(* IEC 61131-3 sources: AXOpen/src/components.cognex.vision/app/src/IO/PLC_LINE, 7 files *)

(* ---- HwIdentifiers.st ---- *)
TYPE
    HwIdentifiers : WORD
    (
        PROFINET_IO_System_HwID :=	WORD#256,
        is7600_HwID :=	WORD#259,
        is7600_Acquisition_Control_Acquisition_Control_HwID :=	WORD#269,
        is7600_Acquisition_Status_Acquisition_Status_HwID :=	WORD#265,
        is7600_Command_Control_Command_Control_HwID :=	WORD#266,
        is7600_Inspection_Control_Inspection_Control_HwID :=	WORD#268,
        is7600_Inspection_Status_Inspection_Status_HwID :=	WORD#264,
        is7600_Rack_HwID :=	WORD#260,
        is7600_Result_Data_64_bytes_Results___64_bytes_HwID :=	WORD#262,
        is7600_SoftEvent_Control_SoftEvent_Control_HwID :=	WORD#267,
        is7600_User_Data_64_bytes_User_Data___64_bytes_HwID :=	WORD#263,
        is7600_is7600_HwID :=	WORD#261,
        is7600_is7600_In_Sight_IS79XX_IS75XX_CC_B_HwID :=	WORD#270,
        is7600_is7600_profinet_HwID :=	WORD#257,
        is7600_is7600_profinet_Port_1_HwID :=	WORD#258,
        plc_line_HwID :=	WORD#32,
        plc_line_Rail_0_HwID :=	WORD#297,
        plc_line_plc_line_HwID :=	WORD#48,
        plc_line_plc_line__plc_line_HwID :=	WORD#49,
        plc_line_plc_line_CPU_display_1_HwID :=	WORD#54,
        plc_line_plc_line_CPU_exec_unit_1_HwID :=	WORD#52,
        plc_line_plc_line_Card_reader_writer_1_HwID :=	WORD#51,
        plc_line_plc_line_DP_interface_1_HwID :=	WORD#60,
        plc_line_plc_line_LicenseManager_1_HwID :=	WORD#42,
        plc_line_plc_line_OPC_UA_1_HwID :=	WORD#117,
        plc_line_plc_line_PROFINET_interface_2_HwID :=	WORD#72,
        plc_line_plc_line_PROFINET_interface_2_Port_1_HwID :=	WORD#73,
        plc_line_plc_line_Virtual_communication_interface_HwID :=	WORD#135,
        plc_line_plc_line_plc_line_HwID :=	WORD#50,
        plc_line_plc_line_profinet_x1_HwID :=	WORD#64,
        plc_line_plc_line_profinet_x1_Port1_HwID :=	WORD#65,
        plc_line_plc_line_profinet_x1_Port2_HwID :=	WORD#66,
        reader_st1_HwID :=	WORD#286,
        reader_st1_Acquisition_Control_Acquisition_Control_HwID :=	WORD#295,
        reader_st1_Acquisition_Status_Acquisition_Status_HwID :=	WORD#294,
        reader_st1_Rack_HwID :=	WORD#287,
        reader_st1_Result_Data_128_bytes_Result_Data___128_bytes_HwID :=	WORD#289,
        reader_st1_Results_Control_Results_Control_HwID :=	WORD#293,
        reader_st1_Results_Status_Results_Status_HwID :=	WORD#292,
        reader_st1_Soft_Event_Control_Soft_Event_Control_HwID :=	WORD#291,
        reader_st1_User_Data_128_bytes_User_Data___128_bytes_HwID :=	WORD#290,
        reader_st1_reader_st1_HwID :=	WORD#288,
        reader_st1_reader_st1_DataMan_280_CC_B_HwID :=	WORD#296,
        reader_st1_reader_st1_profinet_HwID :=	WORD#284,
        reader_st1_reader_st1_profinet_Port_1_HwID :=	WORD#285,
        reader_st2_HwID :=	WORD#273,
        reader_st2_Acquisition_Control_Acquisition_Control_HwID :=	WORD#282,
        reader_st2_Acquisition_Status_Acquisition_Status_HwID :=	WORD#281,
        reader_st2_Rack_HwID :=	WORD#274,
        reader_st2_Result_Data_64_bytes_Result_Data___64_bytes_HwID :=	WORD#276,
        reader_st2_Results_Control_Results_Control_HwID :=	WORD#280,
        reader_st2_Results_Status_Results_Status_HwID :=	WORD#279,
        reader_st2_Soft_Event_Control_Soft_Event_Control_HwID :=	WORD#278,
        reader_st2_User_Data_64_bytes_User_Data___64_bytes_HwID :=	WORD#277,
        reader_st2_reader_st2_HwID :=	WORD#275,
        reader_st2_reader_st2_DataMan_300_HwID :=	WORD#283,
        reader_st2_reader_st2_profinet_HwID :=	WORD#271,
        reader_st2_reader_st2_profinet_Port_1_HwID :=	WORD#272,

        NONE := WORD#0
    );
END_TYPE

(* ---- HwInputs.st ---- *)
TYPE
	HwInputs : STRUCT
		_10a1_Acquisition_Status_1 AT %B82 : ARRAY[0..2] OF BYTE;
		_10a1_Results_Status_1 AT %B85 : BYTE;
		_10a1_Soft_Event_Control_1 AT %B86 : BYTE;
		_10a1_Result_Data_128_bytes_1 AT %B87 : ARRAY[0..135] OF BYTE;
		reader_st2_Acquisition_Status_1 AT %B300 : ARRAY[0..2] OF BYTE;
		reader_st2_Results_Status_1 AT %B303 : BYTE;
		reader_st2_Soft_Event_Control_1 AT %B304 : BYTE;
		reader_st2_Result_Data_64_bytes_1 AT %B305 : ARRAY[0..71] OF BYTE;
		// _7600_Acquisition_Status_1 AT %B0 : ARRAY[0..2] OF BYTE;
		// _7600_Inspection_Status_1 AT %B3 : DWORD;
		// _7600_Command_Control_1 AT %B7 : WORD;
		// _7600_SoftEvent_Control_1 AT %B9 : BYTE;
		// _7600_Results_64_bytes_1 AT %B10 : ARRAY[0..67] OF BYTE;
	END_STRUCT;
END_TYPE

(* ---- HwOutputs.st ---- *)
TYPE
	HwOutputs : STRUCT
		_10a1_Acquisition_Control_1 AT %B72 : BYTE;
		_10a1_Results_Control_1 AT %B73 : BYTE;
		_10a1_Soft_Event_Control_1 AT %B74 : BYTE;
		_10a1_User_Data_128_bytes_1 AT %B75 : ARRAY[0..131] OF BYTE;
		reader_st2_Acquisition_Control_1 AT %B300 : BYTE;
		reader_st2_Results_Control_1 AT %B301 : BYTE;
		reader_st2_Soft_Event_Control_1 AT %B302 : BYTE;
		reader_st2_User_Data_64_bytes_1 AT %B303 : ARRAY[0..67] OF BYTE;
		// _7600_Acquisition_Control_1 AT %B0 : BYTE;
		// _7600_Inspection_Control_1 AT %B1 : BYTE;
		// _7600_Command_Control_1 AT %B2 : WORD;
		// _7600_SoftEvent_Control_1 AT %B4 : BYTE;
		// _7600_User_Data_64_bytes_1 AT %B5 : ARRAY[0..63] OF BYTE;
	END_STRUCT;
END_TYPE

(* ---- PlcInputs.st ---- *)
TYPE
	PlcInputs : STRUCT
		_10a1_Acquisition_Status_1 : ARRAY[0..2] OF BYTE;
		_10a1_Results_Status_1 : BYTE;
		_10a1_Soft_Event_Control_1 : BYTE;
		_10a1_Result_Data_128_bytes_1 : ARRAY[0..135] OF BYTE;
		reader_st2_Acquisition_Status_1 : ARRAY[0..2] OF BYTE;
		reader_st2_Results_Status_1 : BYTE;
		reader_st2_Soft_Event_Control_1 : BYTE;
		reader_st2_Result_Data_64_bytes_1 : ARRAY[0..71] OF BYTE;
		// _7600_Acquisition_Status_1 : ARRAY[0..2] OF BYTE;
		// _7600_Inspection_Status_1 : DWORD;
		// _7600_Command_Control_1 : WORD;
		// _7600_SoftEvent_Control_1 : BYTE;
		// _7600_Results_64_bytes_1 : ARRAY[0..67] OF BYTE;
	END_STRUCT;
END_TYPE

(* ---- PlcOutputs.st ---- *)
TYPE
	PlcOutputs : STRUCT
		_10a1_Acquisition_Control_1 : BYTE;
		_10a1_Results_Control_1 : BYTE;
		_10a1_Soft_Event_Control_1 : BYTE;
		_10a1_User_Data_128_bytes_1 : ARRAY[0..131] OF BYTE;
		reader_st2_Acquisition_Control_1 : BYTE;
		reader_st2_Results_Control_1 : BYTE;
		reader_st2_Soft_Event_Control_1 : BYTE;
		reader_st2_User_Data_64_bytes_1 : ARRAY[0..67] OF BYTE;
		// _7600_Acquisition_Control_1 : BYTE;
		// _7600_Inspection_Control_1 : BYTE;
		// _7600_Command_Control_1 : WORD;
		// _7600_SoftEvent_Control_1 : BYTE;
		// _7600_User_Data_64_bytes_1 : ARRAY[0..63] OF BYTE;
	END_STRUCT;
END_TYPE

(* ---- CopyInputs.st ---- *)
FUNCTION CopyInputs
	VAR_EXTERNAL
		HwInputs : HwInputs;
		PlcInputs : PlcInputs;
	END_VAR
	PlcInputs._10a1_Acquisition_Status_1[0] := HwInputs._10a1_Acquisition_Status_1[0];
	PlcInputs._10a1_Acquisition_Status_1[1] := HwInputs._10a1_Acquisition_Status_1[1];
	PlcInputs._10a1_Acquisition_Status_1[2] := HwInputs._10a1_Acquisition_Status_1[2];
	PlcInputs._10a1_Results_Status_1 := HwInputs._10a1_Results_Status_1;
	PlcInputs._10a1_Soft_Event_Control_1 := HwInputs._10a1_Soft_Event_Control_1;
	PlcInputs._10a1_Result_Data_128_bytes_1[0] := HwInputs._10a1_Result_Data_128_bytes_1[0];
	PlcInputs._10a1_Result_Data_128_bytes_1[1] := HwInputs._10a1_Result_Data_128_bytes_1[1];
	PlcInputs._10a1_Result_Data_128_bytes_1[2] := HwInputs._10a1_Result_Data_128_bytes_1[2];
	PlcInputs._10a1_Result_Data_128_bytes_1[3] := HwInputs._10a1_Result_Data_128_bytes_1[3];
	PlcInputs._10a1_Result_Data_128_bytes_1[4] := HwInputs._10a1_Result_Data_128_bytes_1[4];
	PlcInputs._10a1_Result_Data_128_bytes_1[5] := HwInputs._10a1_Result_Data_128_bytes_1[5];
	PlcInputs._10a1_Result_Data_128_bytes_1[6] := HwInputs._10a1_Result_Data_128_bytes_1[6];
	PlcInputs._10a1_Result_Data_128_bytes_1[7] := HwInputs._10a1_Result_Data_128_bytes_1[7];
	PlcInputs._10a1_Result_Data_128_bytes_1[8] := HwInputs._10a1_Result_Data_128_bytes_1[8];
	PlcInputs._10a1_Result_Data_128_bytes_1[9] := HwInputs._10a1_Result_Data_128_bytes_1[9];
	PlcInputs._10a1_Result_Data_128_bytes_1[10] := HwInputs._10a1_Result_Data_128_bytes_1[10];
	PlcInputs._10a1_Result_Data_128_bytes_1[11] := HwInputs._10a1_Result_Data_128_bytes_1[11];
	PlcInputs._10a1_Result_Data_128_bytes_1[12] := HwInputs._10a1_Result_Data_128_bytes_1[12];
	PlcInputs._10a1_Result_Data_128_bytes_1[13] := HwInputs._10a1_Result_Data_128_bytes_1[13];
	PlcInputs._10a1_Result_Data_128_bytes_1[14] := HwInputs._10a1_Result_Data_128_bytes_1[14];
	PlcInputs._10a1_Result_Data_128_bytes_1[15] := HwInputs._10a1_Result_Data_128_bytes_1[15];
	PlcInputs._10a1_Result_Data_128_bytes_1[16] := HwInputs._10a1_Result_Data_128_bytes_1[16];
	PlcInputs._10a1_Result_Data_128_bytes_1[17] := HwInputs._10a1_Result_Data_128_bytes_1[17];
	PlcInputs._10a1_Result_Data_128_bytes_1[18] := HwInputs._10a1_Result_Data_128_bytes_1[18];
	PlcInputs._10a1_Result_Data_128_bytes_1[19] := HwInputs._10a1_Result_Data_128_bytes_1[19];
	PlcInputs._10a1_Result_Data_128_bytes_1[20] := HwInputs._10a1_Result_Data_128_bytes_1[20];
	PlcInputs._10a1_Result_Data_128_bytes_1[21] := HwInputs._10a1_Result_Data_128_bytes_1[21];
	PlcInputs._10a1_Result_Data_128_bytes_1[22] := HwInputs._10a1_Result_Data_128_bytes_1[22];
	PlcInputs._10a1_Result_Data_128_bytes_1[23] := HwInputs._10a1_Result_Data_128_bytes_1[23];
	PlcInputs._10a1_Result_Data_128_bytes_1[24] := HwInputs._10a1_Result_Data_128_bytes_1[24];
	PlcInputs._10a1_Result_Data_128_bytes_1[25] := HwInputs._10a1_Result_Data_128_bytes_1[25];
	PlcInputs._10a1_Result_Data_128_bytes_1[26] := HwInputs._10a1_Result_Data_128_bytes_1[26];
	PlcInputs._10a1_Result_Data_128_bytes_1[27] := HwInputs._10a1_Result_Data_128_bytes_1[27];
	PlcInputs._10a1_Result_Data_128_bytes_1[28] := HwInputs._10a1_Result_Data_128_bytes_1[28];
	PlcInputs._10a1_Result_Data_128_bytes_1[29] := HwInputs._10a1_Result_Data_128_bytes_1[29];
	PlcInputs._10a1_Result_Data_128_bytes_1[30] := HwInputs._10a1_Result_Data_128_bytes_1[30];
	PlcInputs._10a1_Result_Data_128_bytes_1[31] := HwInputs._10a1_Result_Data_128_bytes_1[31];
	PlcInputs._10a1_Result_Data_128_bytes_1[32] := HwInputs._10a1_Result_Data_128_bytes_1[32];
	PlcInputs._10a1_Result_Data_128_bytes_1[33] := HwInputs._10a1_Result_Data_128_bytes_1[33];
	PlcInputs._10a1_Result_Data_128_bytes_1[34] := HwInputs._10a1_Result_Data_128_bytes_1[34];
	PlcInputs._10a1_Result_Data_128_bytes_1[35] := HwInputs._10a1_Result_Data_128_bytes_1[35];
	PlcInputs._10a1_Result_Data_128_bytes_1[36] := HwInputs._10a1_Result_Data_128_bytes_1[36];
	PlcInputs._10a1_Result_Data_128_bytes_1[37] := HwInputs._10a1_Result_Data_128_bytes_1[37];
	PlcInputs._10a1_Result_Data_128_bytes_1[38] := HwInputs._10a1_Result_Data_128_bytes_1[38];
	PlcInputs._10a1_Result_Data_128_bytes_1[39] := HwInputs._10a1_Result_Data_128_bytes_1[39];
	PlcInputs._10a1_Result_Data_128_bytes_1[40] := HwInputs._10a1_Result_Data_128_bytes_1[40];
	PlcInputs._10a1_Result_Data_128_bytes_1[41] := HwInputs._10a1_Result_Data_128_bytes_1[41];
	PlcInputs._10a1_Result_Data_128_bytes_1[42] := HwInputs._10a1_Result_Data_128_bytes_1[42];
	PlcInputs._10a1_Result_Data_128_bytes_1[43] := HwInputs._10a1_Result_Data_128_bytes_1[43];
	PlcInputs._10a1_Result_Data_128_bytes_1[44] := HwInputs._10a1_Result_Data_128_bytes_1[44];
	PlcInputs._10a1_Result_Data_128_bytes_1[45] := HwInputs._10a1_Result_Data_128_bytes_1[45];
	PlcInputs._10a1_Result_Data_128_bytes_1[46] := HwInputs._10a1_Result_Data_128_bytes_1[46];
	PlcInputs._10a1_Result_Data_128_bytes_1[47] := HwInputs._10a1_Result_Data_128_bytes_1[47];
	PlcInputs._10a1_Result_Data_128_bytes_1[48] := HwInputs._10a1_Result_Data_128_bytes_1[48];
	PlcInputs._10a1_Result_Data_128_bytes_1[49] := HwInputs._10a1_Result_Data_128_bytes_1[49];
	PlcInputs._10a1_Result_Data_128_bytes_1[50] := HwInputs._10a1_Result_Data_128_bytes_1[50];
	PlcInputs._10a1_Result_Data_128_bytes_1[51] := HwInputs._10a1_Result_Data_128_bytes_1[51];
	PlcInputs._10a1_Result_Data_128_bytes_1[52] := HwInputs._10a1_Result_Data_128_bytes_1[52];
	PlcInputs._10a1_Result_Data_128_bytes_1[53] := HwInputs._10a1_Result_Data_128_bytes_1[53];
	PlcInputs._10a1_Result_Data_128_bytes_1[54] := HwInputs._10a1_Result_Data_128_bytes_1[54];
	PlcInputs._10a1_Result_Data_128_bytes_1[55] := HwInputs._10a1_Result_Data_128_bytes_1[55];
	PlcInputs._10a1_Result_Data_128_bytes_1[56] := HwInputs._10a1_Result_Data_128_bytes_1[56];
	PlcInputs._10a1_Result_Data_128_bytes_1[57] := HwInputs._10a1_Result_Data_128_bytes_1[57];
	PlcInputs._10a1_Result_Data_128_bytes_1[58] := HwInputs._10a1_Result_Data_128_bytes_1[58];
	PlcInputs._10a1_Result_Data_128_bytes_1[59] := HwInputs._10a1_Result_Data_128_bytes_1[59];
	PlcInputs._10a1_Result_Data_128_bytes_1[60] := HwInputs._10a1_Result_Data_128_bytes_1[60];
	PlcInputs._10a1_Result_Data_128_bytes_1[61] := HwInputs._10a1_Result_Data_128_bytes_1[61];
	PlcInputs._10a1_Result_Data_128_bytes_1[62] := HwInputs._10a1_Result_Data_128_bytes_1[62];
	PlcInputs._10a1_Result_Data_128_bytes_1[63] := HwInputs._10a1_Result_Data_128_bytes_1[63];
	PlcInputs._10a1_Result_Data_128_bytes_1[64] := HwInputs._10a1_Result_Data_128_bytes_1[64];
	PlcInputs._10a1_Result_Data_128_bytes_1[65] := HwInputs._10a1_Result_Data_128_bytes_1[65];
	PlcInputs._10a1_Result_Data_128_bytes_1[66] := HwInputs._10a1_Result_Data_128_bytes_1[66];
	PlcInputs._10a1_Result_Data_128_bytes_1[67] := HwInputs._10a1_Result_Data_128_bytes_1[67];
	PlcInputs._10a1_Result_Data_128_bytes_1[68] := HwInputs._10a1_Result_Data_128_bytes_1[68];
	PlcInputs._10a1_Result_Data_128_bytes_1[69] := HwInputs._10a1_Result_Data_128_bytes_1[69];
	PlcInputs._10a1_Result_Data_128_bytes_1[70] := HwInputs._10a1_Result_Data_128_bytes_1[70];
	PlcInputs._10a1_Result_Data_128_bytes_1[71] := HwInputs._10a1_Result_Data_128_bytes_1[71];
	PlcInputs._10a1_Result_Data_128_bytes_1[72] := HwInputs._10a1_Result_Data_128_bytes_1[72];
	PlcInputs._10a1_Result_Data_128_bytes_1[73] := HwInputs._10a1_Result_Data_128_bytes_1[73];
	PlcInputs._10a1_Result_Data_128_bytes_1[74] := HwInputs._10a1_Result_Data_128_bytes_1[74];
	PlcInputs._10a1_Result_Data_128_bytes_1[75] := HwInputs._10a1_Result_Data_128_bytes_1[75];
	PlcInputs._10a1_Result_Data_128_bytes_1[76] := HwInputs._10a1_Result_Data_128_bytes_1[76];
	PlcInputs._10a1_Result_Data_128_bytes_1[77] := HwInputs._10a1_Result_Data_128_bytes_1[77];
	PlcInputs._10a1_Result_Data_128_bytes_1[78] := HwInputs._10a1_Result_Data_128_bytes_1[78];
	PlcInputs._10a1_Result_Data_128_bytes_1[79] := HwInputs._10a1_Result_Data_128_bytes_1[79];
	PlcInputs._10a1_Result_Data_128_bytes_1[80] := HwInputs._10a1_Result_Data_128_bytes_1[80];
	PlcInputs._10a1_Result_Data_128_bytes_1[81] := HwInputs._10a1_Result_Data_128_bytes_1[81];
	PlcInputs._10a1_Result_Data_128_bytes_1[82] := HwInputs._10a1_Result_Data_128_bytes_1[82];
	PlcInputs._10a1_Result_Data_128_bytes_1[83] := HwInputs._10a1_Result_Data_128_bytes_1[83];
	PlcInputs._10a1_Result_Data_128_bytes_1[84] := HwInputs._10a1_Result_Data_128_bytes_1[84];
	PlcInputs._10a1_Result_Data_128_bytes_1[85] := HwInputs._10a1_Result_Data_128_bytes_1[85];
	PlcInputs._10a1_Result_Data_128_bytes_1[86] := HwInputs._10a1_Result_Data_128_bytes_1[86];
	PlcInputs._10a1_Result_Data_128_bytes_1[87] := HwInputs._10a1_Result_Data_128_bytes_1[87];
	PlcInputs._10a1_Result_Data_128_bytes_1[88] := HwInputs._10a1_Result_Data_128_bytes_1[88];
	PlcInputs._10a1_Result_Data_128_bytes_1[89] := HwInputs._10a1_Result_Data_128_bytes_1[89];
	PlcInputs._10a1_Result_Data_128_bytes_1[90] := HwInputs._10a1_Result_Data_128_bytes_1[90];
	PlcInputs._10a1_Result_Data_128_bytes_1[91] := HwInputs._10a1_Result_Data_128_bytes_1[91];
	PlcInputs._10a1_Result_Data_128_bytes_1[92] := HwInputs._10a1_Result_Data_128_bytes_1[92];
	PlcInputs._10a1_Result_Data_128_bytes_1[93] := HwInputs._10a1_Result_Data_128_bytes_1[93];
	PlcInputs._10a1_Result_Data_128_bytes_1[94] := HwInputs._10a1_Result_Data_128_bytes_1[94];
	PlcInputs._10a1_Result_Data_128_bytes_1[95] := HwInputs._10a1_Result_Data_128_bytes_1[95];
	PlcInputs._10a1_Result_Data_128_bytes_1[96] := HwInputs._10a1_Result_Data_128_bytes_1[96];
	PlcInputs._10a1_Result_Data_128_bytes_1[97] := HwInputs._10a1_Result_Data_128_bytes_1[97];
	PlcInputs._10a1_Result_Data_128_bytes_1[98] := HwInputs._10a1_Result_Data_128_bytes_1[98];
	PlcInputs._10a1_Result_Data_128_bytes_1[99] := HwInputs._10a1_Result_Data_128_bytes_1[99];
	PlcInputs._10a1_Result_Data_128_bytes_1[100] := HwInputs._10a1_Result_Data_128_bytes_1[100];
	PlcInputs._10a1_Result_Data_128_bytes_1[101] := HwInputs._10a1_Result_Data_128_bytes_1[101];
	PlcInputs._10a1_Result_Data_128_bytes_1[102] := HwInputs._10a1_Result_Data_128_bytes_1[102];
	PlcInputs._10a1_Result_Data_128_bytes_1[103] := HwInputs._10a1_Result_Data_128_bytes_1[103];
	PlcInputs._10a1_Result_Data_128_bytes_1[104] := HwInputs._10a1_Result_Data_128_bytes_1[104];
	PlcInputs._10a1_Result_Data_128_bytes_1[105] := HwInputs._10a1_Result_Data_128_bytes_1[105];
	PlcInputs._10a1_Result_Data_128_bytes_1[106] := HwInputs._10a1_Result_Data_128_bytes_1[106];
	PlcInputs._10a1_Result_Data_128_bytes_1[107] := HwInputs._10a1_Result_Data_128_bytes_1[107];
	PlcInputs._10a1_Result_Data_128_bytes_1[108] := HwInputs._10a1_Result_Data_128_bytes_1[108];
	PlcInputs._10a1_Result_Data_128_bytes_1[109] := HwInputs._10a1_Result_Data_128_bytes_1[109];
	PlcInputs._10a1_Result_Data_128_bytes_1[110] := HwInputs._10a1_Result_Data_128_bytes_1[110];
	PlcInputs._10a1_Result_Data_128_bytes_1[111] := HwInputs._10a1_Result_Data_128_bytes_1[111];
	PlcInputs._10a1_Result_Data_128_bytes_1[112] := HwInputs._10a1_Result_Data_128_bytes_1[112];
	PlcInputs._10a1_Result_Data_128_bytes_1[113] := HwInputs._10a1_Result_Data_128_bytes_1[113];
	PlcInputs._10a1_Result_Data_128_bytes_1[114] := HwInputs._10a1_Result_Data_128_bytes_1[114];
	PlcInputs._10a1_Result_Data_128_bytes_1[115] := HwInputs._10a1_Result_Data_128_bytes_1[115];
	PlcInputs._10a1_Result_Data_128_bytes_1[116] := HwInputs._10a1_Result_Data_128_bytes_1[116];
	PlcInputs._10a1_Result_Data_128_bytes_1[117] := HwInputs._10a1_Result_Data_128_bytes_1[117];
	PlcInputs._10a1_Result_Data_128_bytes_1[118] := HwInputs._10a1_Result_Data_128_bytes_1[118];
	PlcInputs._10a1_Result_Data_128_bytes_1[119] := HwInputs._10a1_Result_Data_128_bytes_1[119];
	PlcInputs._10a1_Result_Data_128_bytes_1[120] := HwInputs._10a1_Result_Data_128_bytes_1[120];
	PlcInputs._10a1_Result_Data_128_bytes_1[121] := HwInputs._10a1_Result_Data_128_bytes_1[121];
	PlcInputs._10a1_Result_Data_128_bytes_1[122] := HwInputs._10a1_Result_Data_128_bytes_1[122];
	PlcInputs._10a1_Result_Data_128_bytes_1[123] := HwInputs._10a1_Result_Data_128_bytes_1[123];
	PlcInputs._10a1_Result_Data_128_bytes_1[124] := HwInputs._10a1_Result_Data_128_bytes_1[124];
	PlcInputs._10a1_Result_Data_128_bytes_1[125] := HwInputs._10a1_Result_Data_128_bytes_1[125];
	PlcInputs._10a1_Result_Data_128_bytes_1[126] := HwInputs._10a1_Result_Data_128_bytes_1[126];
	PlcInputs._10a1_Result_Data_128_bytes_1[127] := HwInputs._10a1_Result_Data_128_bytes_1[127];
	PlcInputs._10a1_Result_Data_128_bytes_1[128] := HwInputs._10a1_Result_Data_128_bytes_1[128];
	PlcInputs._10a1_Result_Data_128_bytes_1[129] := HwInputs._10a1_Result_Data_128_bytes_1[129];
	PlcInputs._10a1_Result_Data_128_bytes_1[130] := HwInputs._10a1_Result_Data_128_bytes_1[130];
	PlcInputs._10a1_Result_Data_128_bytes_1[131] := HwInputs._10a1_Result_Data_128_bytes_1[131];
	PlcInputs._10a1_Result_Data_128_bytes_1[132] := HwInputs._10a1_Result_Data_128_bytes_1[132];
	PlcInputs._10a1_Result_Data_128_bytes_1[133] := HwInputs._10a1_Result_Data_128_bytes_1[133];
	PlcInputs._10a1_Result_Data_128_bytes_1[134] := HwInputs._10a1_Result_Data_128_bytes_1[134];
	PlcInputs._10a1_Result_Data_128_bytes_1[135] := HwInputs._10a1_Result_Data_128_bytes_1[135];
	PlcInputs.reader_st2_Acquisition_Status_1[0] := HwInputs.reader_st2_Acquisition_Status_1[0];
	PlcInputs.reader_st2_Acquisition_Status_1[1] := HwInputs.reader_st2_Acquisition_Status_1[1];
	PlcInputs.reader_st2_Acquisition_Status_1[2] := HwInputs.reader_st2_Acquisition_Status_1[2];
	PlcInputs.reader_st2_Results_Status_1 := HwInputs.reader_st2_Results_Status_1;
	PlcInputs.reader_st2_Soft_Event_Control_1 := HwInputs.reader_st2_Soft_Event_Control_1;
	PlcInputs.reader_st2_Result_Data_64_bytes_1[0] := HwInputs.reader_st2_Result_Data_64_bytes_1[0];
	PlcInputs.reader_st2_Result_Data_64_bytes_1[1] := HwInputs.reader_st2_Result_Data_64_bytes_1[1];
	PlcInputs.reader_st2_Result_Data_64_bytes_1[2] := HwInputs.reader_st2_Result_Data_64_bytes_1[2];
	PlcInputs.reader_st2_Result_Data_64_bytes_1[3] := HwInputs.reader_st2_Result_Data_64_bytes_1[3];
	PlcInputs.reader_st2_Result_Data_64_bytes_1[4] := HwInputs.reader_st2_Result_Data_64_bytes_1[4];
	PlcInputs.reader_st2_Result_Data_64_bytes_1[5] := HwInputs.reader_st2_Result_Data_64_bytes_1[5];
	PlcInputs.reader_st2_Result_Data_64_bytes_1[6] := HwInputs.reader_st2_Result_Data_64_bytes_1[6];
	PlcInputs.reader_st2_Result_Data_64_bytes_1[7] := HwInputs.reader_st2_Result_Data_64_bytes_1[7];
	PlcInputs.reader_st2_Result_Data_64_bytes_1[8] := HwInputs.reader_st2_Result_Data_64_bytes_1[8];
	PlcInputs.reader_st2_Result_Data_64_bytes_1[9] := HwInputs.reader_st2_Result_Data_64_bytes_1[9];
	PlcInputs.reader_st2_Result_Data_64_bytes_1[10] := HwInputs.reader_st2_Result_Data_64_bytes_1[10];
	PlcInputs.reader_st2_Result_Data_64_bytes_1[11] := HwInputs.reader_st2_Result_Data_64_bytes_1[11];
	PlcInputs.reader_st2_Result_Data_64_bytes_1[12] := HwInputs.reader_st2_Result_Data_64_bytes_1[12];
	PlcInputs.reader_st2_Result_Data_64_bytes_1[13] := HwInputs.reader_st2_Result_Data_64_bytes_1[13];
	PlcInputs.reader_st2_Result_Data_64_bytes_1[14] := HwInputs.reader_st2_Result_Data_64_bytes_1[14];
	PlcInputs.reader_st2_Result_Data_64_bytes_1[15] := HwInputs.reader_st2_Result_Data_64_bytes_1[15];
	PlcInputs.reader_st2_Result_Data_64_bytes_1[16] := HwInputs.reader_st2_Result_Data_64_bytes_1[16];
	PlcInputs.reader_st2_Result_Data_64_bytes_1[17] := HwInputs.reader_st2_Result_Data_64_bytes_1[17];
	PlcInputs.reader_st2_Result_Data_64_bytes_1[18] := HwInputs.reader_st2_Result_Data_64_bytes_1[18];
	PlcInputs.reader_st2_Result_Data_64_bytes_1[19] := HwInputs.reader_st2_Result_Data_64_bytes_1[19];
	PlcInputs.reader_st2_Result_Data_64_bytes_1[20] := HwInputs.reader_st2_Result_Data_64_bytes_1[20];
	PlcInputs.reader_st2_Result_Data_64_bytes_1[21] := HwInputs.reader_st2_Result_Data_64_bytes_1[21];
	PlcInputs.reader_st2_Result_Data_64_bytes_1[22] := HwInputs.reader_st2_Result_Data_64_bytes_1[22];
	PlcInputs.reader_st2_Result_Data_64_bytes_1[23] := HwInputs.reader_st2_Result_Data_64_bytes_1[23];
	PlcInputs.reader_st2_Result_Data_64_bytes_1[24] := HwInputs.reader_st2_Result_Data_64_bytes_1[24];
	PlcInputs.reader_st2_Result_Data_64_bytes_1[25] := HwInputs.reader_st2_Result_Data_64_bytes_1[25];
	PlcInputs.reader_st2_Result_Data_64_bytes_1[26] := HwInputs.reader_st2_Result_Data_64_bytes_1[26];
	PlcInputs.reader_st2_Result_Data_64_bytes_1[27] := HwInputs.reader_st2_Result_Data_64_bytes_1[27];
	PlcInputs.reader_st2_Result_Data_64_bytes_1[28] := HwInputs.reader_st2_Result_Data_64_bytes_1[28];
	PlcInputs.reader_st2_Result_Data_64_bytes_1[29] := HwInputs.reader_st2_Result_Data_64_bytes_1[29];
	PlcInputs.reader_st2_Result_Data_64_bytes_1[30] := HwInputs.reader_st2_Result_Data_64_bytes_1[30];
	PlcInputs.reader_st2_Result_Data_64_bytes_1[31] := HwInputs.reader_st2_Result_Data_64_bytes_1[31];
	PlcInputs.reader_st2_Result_Data_64_bytes_1[32] := HwInputs.reader_st2_Result_Data_64_bytes_1[32];
	PlcInputs.reader_st2_Result_Data_64_bytes_1[33] := HwInputs.reader_st2_Result_Data_64_bytes_1[33];
	PlcInputs.reader_st2_Result_Data_64_bytes_1[34] := HwInputs.reader_st2_Result_Data_64_bytes_1[34];
	PlcInputs.reader_st2_Result_Data_64_bytes_1[35] := HwInputs.reader_st2_Result_Data_64_bytes_1[35];
	PlcInputs.reader_st2_Result_Data_64_bytes_1[36] := HwInputs.reader_st2_Result_Data_64_bytes_1[36];
	PlcInputs.reader_st2_Result_Data_64_bytes_1[37] := HwInputs.reader_st2_Result_Data_64_bytes_1[37];
	PlcInputs.reader_st2_Result_Data_64_bytes_1[38] := HwInputs.reader_st2_Result_Data_64_bytes_1[38];
	PlcInputs.reader_st2_Result_Data_64_bytes_1[39] := HwInputs.reader_st2_Result_Data_64_bytes_1[39];
	PlcInputs.reader_st2_Result_Data_64_bytes_1[40] := HwInputs.reader_st2_Result_Data_64_bytes_1[40];
	PlcInputs.reader_st2_Result_Data_64_bytes_1[41] := HwInputs.reader_st2_Result_Data_64_bytes_1[41];
	PlcInputs.reader_st2_Result_Data_64_bytes_1[42] := HwInputs.reader_st2_Result_Data_64_bytes_1[42];
	PlcInputs.reader_st2_Result_Data_64_bytes_1[43] := HwInputs.reader_st2_Result_Data_64_bytes_1[43];
	PlcInputs.reader_st2_Result_Data_64_bytes_1[44] := HwInputs.reader_st2_Result_Data_64_bytes_1[44];
	PlcInputs.reader_st2_Result_Data_64_bytes_1[45] := HwInputs.reader_st2_Result_Data_64_bytes_1[45];
	PlcInputs.reader_st2_Result_Data_64_bytes_1[46] := HwInputs.reader_st2_Result_Data_64_bytes_1[46];
	PlcInputs.reader_st2_Result_Data_64_bytes_1[47] := HwInputs.reader_st2_Result_Data_64_bytes_1[47];
	PlcInputs.reader_st2_Result_Data_64_bytes_1[48] := HwInputs.reader_st2_Result_Data_64_bytes_1[48];
	PlcInputs.reader_st2_Result_Data_64_bytes_1[49] := HwInputs.reader_st2_Result_Data_64_bytes_1[49];
	PlcInputs.reader_st2_Result_Data_64_bytes_1[50] := HwInputs.reader_st2_Result_Data_64_bytes_1[50];
	PlcInputs.reader_st2_Result_Data_64_bytes_1[51] := HwInputs.reader_st2_Result_Data_64_bytes_1[51];
	PlcInputs.reader_st2_Result_Data_64_bytes_1[52] := HwInputs.reader_st2_Result_Data_64_bytes_1[52];
	PlcInputs.reader_st2_Result_Data_64_bytes_1[53] := HwInputs.reader_st2_Result_Data_64_bytes_1[53];
	PlcInputs.reader_st2_Result_Data_64_bytes_1[54] := HwInputs.reader_st2_Result_Data_64_bytes_1[54];
	PlcInputs.reader_st2_Result_Data_64_bytes_1[55] := HwInputs.reader_st2_Result_Data_64_bytes_1[55];
	PlcInputs.reader_st2_Result_Data_64_bytes_1[56] := HwInputs.reader_st2_Result_Data_64_bytes_1[56];
	PlcInputs.reader_st2_Result_Data_64_bytes_1[57] := HwInputs.reader_st2_Result_Data_64_bytes_1[57];
	PlcInputs.reader_st2_Result_Data_64_bytes_1[58] := HwInputs.reader_st2_Result_Data_64_bytes_1[58];
	PlcInputs.reader_st2_Result_Data_64_bytes_1[59] := HwInputs.reader_st2_Result_Data_64_bytes_1[59];
	PlcInputs.reader_st2_Result_Data_64_bytes_1[60] := HwInputs.reader_st2_Result_Data_64_bytes_1[60];
	PlcInputs.reader_st2_Result_Data_64_bytes_1[61] := HwInputs.reader_st2_Result_Data_64_bytes_1[61];
	PlcInputs.reader_st2_Result_Data_64_bytes_1[62] := HwInputs.reader_st2_Result_Data_64_bytes_1[62];
	PlcInputs.reader_st2_Result_Data_64_bytes_1[63] := HwInputs.reader_st2_Result_Data_64_bytes_1[63];
	PlcInputs.reader_st2_Result_Data_64_bytes_1[64] := HwInputs.reader_st2_Result_Data_64_bytes_1[64];
	PlcInputs.reader_st2_Result_Data_64_bytes_1[65] := HwInputs.reader_st2_Result_Data_64_bytes_1[65];
	PlcInputs.reader_st2_Result_Data_64_bytes_1[66] := HwInputs.reader_st2_Result_Data_64_bytes_1[66];
	PlcInputs.reader_st2_Result_Data_64_bytes_1[67] := HwInputs.reader_st2_Result_Data_64_bytes_1[67];
	PlcInputs.reader_st2_Result_Data_64_bytes_1[68] := HwInputs.reader_st2_Result_Data_64_bytes_1[68];
	PlcInputs.reader_st2_Result_Data_64_bytes_1[69] := HwInputs.reader_st2_Result_Data_64_bytes_1[69];
	PlcInputs.reader_st2_Result_Data_64_bytes_1[70] := HwInputs.reader_st2_Result_Data_64_bytes_1[70];
	PlcInputs.reader_st2_Result_Data_64_bytes_1[71] := HwInputs.reader_st2_Result_Data_64_bytes_1[71];
	// PlcInputs._7600_Acquisition_Status_1[0] := HwInputs._7600_Acquisition_Status_1[0];
	// PlcInputs._7600_Acquisition_Status_1[1] := HwInputs._7600_Acquisition_Status_1[1];
	// PlcInputs._7600_Acquisition_Status_1[2] := HwInputs._7600_Acquisition_Status_1[2];
	// PlcInputs._7600_Inspection_Status_1 := HwInputs._7600_Inspection_Status_1;
	// PlcInputs._7600_Command_Control_1 := HwInputs._7600_Command_Control_1;
	// PlcInputs._7600_SoftEvent_Control_1 := HwInputs._7600_SoftEvent_Control_1;
	// PlcInputs._7600_Results_64_bytes_1[0] := HwInputs._7600_Results_64_bytes_1[0];
	// PlcInputs._7600_Results_64_bytes_1[1] := HwInputs._7600_Results_64_bytes_1[1];
	// PlcInputs._7600_Results_64_bytes_1[2] := HwInputs._7600_Results_64_bytes_1[2];
	// PlcInputs._7600_Results_64_bytes_1[3] := HwInputs._7600_Results_64_bytes_1[3];
	// PlcInputs._7600_Results_64_bytes_1[4] := HwInputs._7600_Results_64_bytes_1[4];
	// PlcInputs._7600_Results_64_bytes_1[5] := HwInputs._7600_Results_64_bytes_1[5];
	// PlcInputs._7600_Results_64_bytes_1[6] := HwInputs._7600_Results_64_bytes_1[6];
	// PlcInputs._7600_Results_64_bytes_1[7] := HwInputs._7600_Results_64_bytes_1[7];
	// PlcInputs._7600_Results_64_bytes_1[8] := HwInputs._7600_Results_64_bytes_1[8];
	// PlcInputs._7600_Results_64_bytes_1[9] := HwInputs._7600_Results_64_bytes_1[9];
	// PlcInputs._7600_Results_64_bytes_1[10] := HwInputs._7600_Results_64_bytes_1[10];
	// PlcInputs._7600_Results_64_bytes_1[11] := HwInputs._7600_Results_64_bytes_1[11];
	// PlcInputs._7600_Results_64_bytes_1[12] := HwInputs._7600_Results_64_bytes_1[12];
	// PlcInputs._7600_Results_64_bytes_1[13] := HwInputs._7600_Results_64_bytes_1[13];
	// PlcInputs._7600_Results_64_bytes_1[14] := HwInputs._7600_Results_64_bytes_1[14];
	// PlcInputs._7600_Results_64_bytes_1[15] := HwInputs._7600_Results_64_bytes_1[15];
	// PlcInputs._7600_Results_64_bytes_1[16] := HwInputs._7600_Results_64_bytes_1[16];
	// PlcInputs._7600_Results_64_bytes_1[17] := HwInputs._7600_Results_64_bytes_1[17];
	// PlcInputs._7600_Results_64_bytes_1[18] := HwInputs._7600_Results_64_bytes_1[18];
	// PlcInputs._7600_Results_64_bytes_1[19] := HwInputs._7600_Results_64_bytes_1[19];
	// PlcInputs._7600_Results_64_bytes_1[20] := HwInputs._7600_Results_64_bytes_1[20];
	// PlcInputs._7600_Results_64_bytes_1[21] := HwInputs._7600_Results_64_bytes_1[21];
	// PlcInputs._7600_Results_64_bytes_1[22] := HwInputs._7600_Results_64_bytes_1[22];
	// PlcInputs._7600_Results_64_bytes_1[23] := HwInputs._7600_Results_64_bytes_1[23];
	// PlcInputs._7600_Results_64_bytes_1[24] := HwInputs._7600_Results_64_bytes_1[24];
	// PlcInputs._7600_Results_64_bytes_1[25] := HwInputs._7600_Results_64_bytes_1[25];
	// PlcInputs._7600_Results_64_bytes_1[26] := HwInputs._7600_Results_64_bytes_1[26];
	// PlcInputs._7600_Results_64_bytes_1[27] := HwInputs._7600_Results_64_bytes_1[27];
	// PlcInputs._7600_Results_64_bytes_1[28] := HwInputs._7600_Results_64_bytes_1[28];
	// PlcInputs._7600_Results_64_bytes_1[29] := HwInputs._7600_Results_64_bytes_1[29];
	// PlcInputs._7600_Results_64_bytes_1[30] := HwInputs._7600_Results_64_bytes_1[30];
	// PlcInputs._7600_Results_64_bytes_1[31] := HwInputs._7600_Results_64_bytes_1[31];
	// PlcInputs._7600_Results_64_bytes_1[32] := HwInputs._7600_Results_64_bytes_1[32];
	// PlcInputs._7600_Results_64_bytes_1[33] := HwInputs._7600_Results_64_bytes_1[33];
	// PlcInputs._7600_Results_64_bytes_1[34] := HwInputs._7600_Results_64_bytes_1[34];
	// PlcInputs._7600_Results_64_bytes_1[35] := HwInputs._7600_Results_64_bytes_1[35];
	// PlcInputs._7600_Results_64_bytes_1[36] := HwInputs._7600_Results_64_bytes_1[36];
	// PlcInputs._7600_Results_64_bytes_1[37] := HwInputs._7600_Results_64_bytes_1[37];
	// PlcInputs._7600_Results_64_bytes_1[38] := HwInputs._7600_Results_64_bytes_1[38];
	// PlcInputs._7600_Results_64_bytes_1[39] := HwInputs._7600_Results_64_bytes_1[39];
	// PlcInputs._7600_Results_64_bytes_1[40] := HwInputs._7600_Results_64_bytes_1[40];
	// PlcInputs._7600_Results_64_bytes_1[41] := HwInputs._7600_Results_64_bytes_1[41];
	// PlcInputs._7600_Results_64_bytes_1[42] := HwInputs._7600_Results_64_bytes_1[42];
	// PlcInputs._7600_Results_64_bytes_1[43] := HwInputs._7600_Results_64_bytes_1[43];
	// PlcInputs._7600_Results_64_bytes_1[44] := HwInputs._7600_Results_64_bytes_1[44];
	// PlcInputs._7600_Results_64_bytes_1[45] := HwInputs._7600_Results_64_bytes_1[45];
	// PlcInputs._7600_Results_64_bytes_1[46] := HwInputs._7600_Results_64_bytes_1[46];
	// PlcInputs._7600_Results_64_bytes_1[47] := HwInputs._7600_Results_64_bytes_1[47];
	// PlcInputs._7600_Results_64_bytes_1[48] := HwInputs._7600_Results_64_bytes_1[48];
	// PlcInputs._7600_Results_64_bytes_1[49] := HwInputs._7600_Results_64_bytes_1[49];
	// PlcInputs._7600_Results_64_bytes_1[50] := HwInputs._7600_Results_64_bytes_1[50];
	// PlcInputs._7600_Results_64_bytes_1[51] := HwInputs._7600_Results_64_bytes_1[51];
	// PlcInputs._7600_Results_64_bytes_1[52] := HwInputs._7600_Results_64_bytes_1[52];
	// PlcInputs._7600_Results_64_bytes_1[53] := HwInputs._7600_Results_64_bytes_1[53];
	// PlcInputs._7600_Results_64_bytes_1[54] := HwInputs._7600_Results_64_bytes_1[54];
	// PlcInputs._7600_Results_64_bytes_1[55] := HwInputs._7600_Results_64_bytes_1[55];
	// PlcInputs._7600_Results_64_bytes_1[56] := HwInputs._7600_Results_64_bytes_1[56];
	// PlcInputs._7600_Results_64_bytes_1[57] := HwInputs._7600_Results_64_bytes_1[57];
	// PlcInputs._7600_Results_64_bytes_1[58] := HwInputs._7600_Results_64_bytes_1[58];
	// PlcInputs._7600_Results_64_bytes_1[59] := HwInputs._7600_Results_64_bytes_1[59];
	// PlcInputs._7600_Results_64_bytes_1[60] := HwInputs._7600_Results_64_bytes_1[60];
	// PlcInputs._7600_Results_64_bytes_1[61] := HwInputs._7600_Results_64_bytes_1[61];
	// PlcInputs._7600_Results_64_bytes_1[62] := HwInputs._7600_Results_64_bytes_1[62];
	// PlcInputs._7600_Results_64_bytes_1[63] := HwInputs._7600_Results_64_bytes_1[63];
	// PlcInputs._7600_Results_64_bytes_1[64] := HwInputs._7600_Results_64_bytes_1[64];
	// PlcInputs._7600_Results_64_bytes_1[65] := HwInputs._7600_Results_64_bytes_1[65];
	// PlcInputs._7600_Results_64_bytes_1[66] := HwInputs._7600_Results_64_bytes_1[66];
	// PlcInputs._7600_Results_64_bytes_1[67] := HwInputs._7600_Results_64_bytes_1[67];
END_FUNCTION

(* ---- CopyOutputs.st ---- *)
FUNCTION CopyOutputs
	VAR_EXTERNAL
		HwOutputs : HwOutputs;
		PlcOutputs : PlcOutputs;
	END_VAR
	HwOutputs._10a1_Acquisition_Control_1 := PlcOutputs._10a1_Acquisition_Control_1;
	HwOutputs._10a1_Results_Control_1 := PlcOutputs._10a1_Results_Control_1;
	HwOutputs._10a1_Soft_Event_Control_1 := PlcOutputs._10a1_Soft_Event_Control_1;
	HwOutputs._10a1_User_Data_128_bytes_1[0] := PlcOutputs._10a1_User_Data_128_bytes_1[0];
	HwOutputs._10a1_User_Data_128_bytes_1[1] := PlcOutputs._10a1_User_Data_128_bytes_1[1];
	HwOutputs._10a1_User_Data_128_bytes_1[2] := PlcOutputs._10a1_User_Data_128_bytes_1[2];
	HwOutputs._10a1_User_Data_128_bytes_1[3] := PlcOutputs._10a1_User_Data_128_bytes_1[3];
	HwOutputs._10a1_User_Data_128_bytes_1[4] := PlcOutputs._10a1_User_Data_128_bytes_1[4];
	HwOutputs._10a1_User_Data_128_bytes_1[5] := PlcOutputs._10a1_User_Data_128_bytes_1[5];
	HwOutputs._10a1_User_Data_128_bytes_1[6] := PlcOutputs._10a1_User_Data_128_bytes_1[6];
	HwOutputs._10a1_User_Data_128_bytes_1[7] := PlcOutputs._10a1_User_Data_128_bytes_1[7];
	HwOutputs._10a1_User_Data_128_bytes_1[8] := PlcOutputs._10a1_User_Data_128_bytes_1[8];
	HwOutputs._10a1_User_Data_128_bytes_1[9] := PlcOutputs._10a1_User_Data_128_bytes_1[9];
	HwOutputs._10a1_User_Data_128_bytes_1[10] := PlcOutputs._10a1_User_Data_128_bytes_1[10];
	HwOutputs._10a1_User_Data_128_bytes_1[11] := PlcOutputs._10a1_User_Data_128_bytes_1[11];
	HwOutputs._10a1_User_Data_128_bytes_1[12] := PlcOutputs._10a1_User_Data_128_bytes_1[12];
	HwOutputs._10a1_User_Data_128_bytes_1[13] := PlcOutputs._10a1_User_Data_128_bytes_1[13];
	HwOutputs._10a1_User_Data_128_bytes_1[14] := PlcOutputs._10a1_User_Data_128_bytes_1[14];
	HwOutputs._10a1_User_Data_128_bytes_1[15] := PlcOutputs._10a1_User_Data_128_bytes_1[15];
	HwOutputs._10a1_User_Data_128_bytes_1[16] := PlcOutputs._10a1_User_Data_128_bytes_1[16];
	HwOutputs._10a1_User_Data_128_bytes_1[17] := PlcOutputs._10a1_User_Data_128_bytes_1[17];
	HwOutputs._10a1_User_Data_128_bytes_1[18] := PlcOutputs._10a1_User_Data_128_bytes_1[18];
	HwOutputs._10a1_User_Data_128_bytes_1[19] := PlcOutputs._10a1_User_Data_128_bytes_1[19];
	HwOutputs._10a1_User_Data_128_bytes_1[20] := PlcOutputs._10a1_User_Data_128_bytes_1[20];
	HwOutputs._10a1_User_Data_128_bytes_1[21] := PlcOutputs._10a1_User_Data_128_bytes_1[21];
	HwOutputs._10a1_User_Data_128_bytes_1[22] := PlcOutputs._10a1_User_Data_128_bytes_1[22];
	HwOutputs._10a1_User_Data_128_bytes_1[23] := PlcOutputs._10a1_User_Data_128_bytes_1[23];
	HwOutputs._10a1_User_Data_128_bytes_1[24] := PlcOutputs._10a1_User_Data_128_bytes_1[24];
	HwOutputs._10a1_User_Data_128_bytes_1[25] := PlcOutputs._10a1_User_Data_128_bytes_1[25];
	HwOutputs._10a1_User_Data_128_bytes_1[26] := PlcOutputs._10a1_User_Data_128_bytes_1[26];
	HwOutputs._10a1_User_Data_128_bytes_1[27] := PlcOutputs._10a1_User_Data_128_bytes_1[27];
	HwOutputs._10a1_User_Data_128_bytes_1[28] := PlcOutputs._10a1_User_Data_128_bytes_1[28];
	HwOutputs._10a1_User_Data_128_bytes_1[29] := PlcOutputs._10a1_User_Data_128_bytes_1[29];
	HwOutputs._10a1_User_Data_128_bytes_1[30] := PlcOutputs._10a1_User_Data_128_bytes_1[30];
	HwOutputs._10a1_User_Data_128_bytes_1[31] := PlcOutputs._10a1_User_Data_128_bytes_1[31];
	HwOutputs._10a1_User_Data_128_bytes_1[32] := PlcOutputs._10a1_User_Data_128_bytes_1[32];
	HwOutputs._10a1_User_Data_128_bytes_1[33] := PlcOutputs._10a1_User_Data_128_bytes_1[33];
	HwOutputs._10a1_User_Data_128_bytes_1[34] := PlcOutputs._10a1_User_Data_128_bytes_1[34];
	HwOutputs._10a1_User_Data_128_bytes_1[35] := PlcOutputs._10a1_User_Data_128_bytes_1[35];
	HwOutputs._10a1_User_Data_128_bytes_1[36] := PlcOutputs._10a1_User_Data_128_bytes_1[36];
	HwOutputs._10a1_User_Data_128_bytes_1[37] := PlcOutputs._10a1_User_Data_128_bytes_1[37];
	HwOutputs._10a1_User_Data_128_bytes_1[38] := PlcOutputs._10a1_User_Data_128_bytes_1[38];
	HwOutputs._10a1_User_Data_128_bytes_1[39] := PlcOutputs._10a1_User_Data_128_bytes_1[39];
	HwOutputs._10a1_User_Data_128_bytes_1[40] := PlcOutputs._10a1_User_Data_128_bytes_1[40];
	HwOutputs._10a1_User_Data_128_bytes_1[41] := PlcOutputs._10a1_User_Data_128_bytes_1[41];
	HwOutputs._10a1_User_Data_128_bytes_1[42] := PlcOutputs._10a1_User_Data_128_bytes_1[42];
	HwOutputs._10a1_User_Data_128_bytes_1[43] := PlcOutputs._10a1_User_Data_128_bytes_1[43];
	HwOutputs._10a1_User_Data_128_bytes_1[44] := PlcOutputs._10a1_User_Data_128_bytes_1[44];
	HwOutputs._10a1_User_Data_128_bytes_1[45] := PlcOutputs._10a1_User_Data_128_bytes_1[45];
	HwOutputs._10a1_User_Data_128_bytes_1[46] := PlcOutputs._10a1_User_Data_128_bytes_1[46];
	HwOutputs._10a1_User_Data_128_bytes_1[47] := PlcOutputs._10a1_User_Data_128_bytes_1[47];
	HwOutputs._10a1_User_Data_128_bytes_1[48] := PlcOutputs._10a1_User_Data_128_bytes_1[48];
	HwOutputs._10a1_User_Data_128_bytes_1[49] := PlcOutputs._10a1_User_Data_128_bytes_1[49];
	HwOutputs._10a1_User_Data_128_bytes_1[50] := PlcOutputs._10a1_User_Data_128_bytes_1[50];
	HwOutputs._10a1_User_Data_128_bytes_1[51] := PlcOutputs._10a1_User_Data_128_bytes_1[51];
	HwOutputs._10a1_User_Data_128_bytes_1[52] := PlcOutputs._10a1_User_Data_128_bytes_1[52];
	HwOutputs._10a1_User_Data_128_bytes_1[53] := PlcOutputs._10a1_User_Data_128_bytes_1[53];
	HwOutputs._10a1_User_Data_128_bytes_1[54] := PlcOutputs._10a1_User_Data_128_bytes_1[54];
	HwOutputs._10a1_User_Data_128_bytes_1[55] := PlcOutputs._10a1_User_Data_128_bytes_1[55];
	HwOutputs._10a1_User_Data_128_bytes_1[56] := PlcOutputs._10a1_User_Data_128_bytes_1[56];
	HwOutputs._10a1_User_Data_128_bytes_1[57] := PlcOutputs._10a1_User_Data_128_bytes_1[57];
	HwOutputs._10a1_User_Data_128_bytes_1[58] := PlcOutputs._10a1_User_Data_128_bytes_1[58];
	HwOutputs._10a1_User_Data_128_bytes_1[59] := PlcOutputs._10a1_User_Data_128_bytes_1[59];
	HwOutputs._10a1_User_Data_128_bytes_1[60] := PlcOutputs._10a1_User_Data_128_bytes_1[60];
	HwOutputs._10a1_User_Data_128_bytes_1[61] := PlcOutputs._10a1_User_Data_128_bytes_1[61];
	HwOutputs._10a1_User_Data_128_bytes_1[62] := PlcOutputs._10a1_User_Data_128_bytes_1[62];
	HwOutputs._10a1_User_Data_128_bytes_1[63] := PlcOutputs._10a1_User_Data_128_bytes_1[63];
	HwOutputs._10a1_User_Data_128_bytes_1[64] := PlcOutputs._10a1_User_Data_128_bytes_1[64];
	HwOutputs._10a1_User_Data_128_bytes_1[65] := PlcOutputs._10a1_User_Data_128_bytes_1[65];
	HwOutputs._10a1_User_Data_128_bytes_1[66] := PlcOutputs._10a1_User_Data_128_bytes_1[66];
	HwOutputs._10a1_User_Data_128_bytes_1[67] := PlcOutputs._10a1_User_Data_128_bytes_1[67];
	HwOutputs._10a1_User_Data_128_bytes_1[68] := PlcOutputs._10a1_User_Data_128_bytes_1[68];
	HwOutputs._10a1_User_Data_128_bytes_1[69] := PlcOutputs._10a1_User_Data_128_bytes_1[69];
	HwOutputs._10a1_User_Data_128_bytes_1[70] := PlcOutputs._10a1_User_Data_128_bytes_1[70];
	HwOutputs._10a1_User_Data_128_bytes_1[71] := PlcOutputs._10a1_User_Data_128_bytes_1[71];
	HwOutputs._10a1_User_Data_128_bytes_1[72] := PlcOutputs._10a1_User_Data_128_bytes_1[72];
	HwOutputs._10a1_User_Data_128_bytes_1[73] := PlcOutputs._10a1_User_Data_128_bytes_1[73];
	HwOutputs._10a1_User_Data_128_bytes_1[74] := PlcOutputs._10a1_User_Data_128_bytes_1[74];
	HwOutputs._10a1_User_Data_128_bytes_1[75] := PlcOutputs._10a1_User_Data_128_bytes_1[75];
	HwOutputs._10a1_User_Data_128_bytes_1[76] := PlcOutputs._10a1_User_Data_128_bytes_1[76];
	HwOutputs._10a1_User_Data_128_bytes_1[77] := PlcOutputs._10a1_User_Data_128_bytes_1[77];
	HwOutputs._10a1_User_Data_128_bytes_1[78] := PlcOutputs._10a1_User_Data_128_bytes_1[78];
	HwOutputs._10a1_User_Data_128_bytes_1[79] := PlcOutputs._10a1_User_Data_128_bytes_1[79];
	HwOutputs._10a1_User_Data_128_bytes_1[80] := PlcOutputs._10a1_User_Data_128_bytes_1[80];
	HwOutputs._10a1_User_Data_128_bytes_1[81] := PlcOutputs._10a1_User_Data_128_bytes_1[81];
	HwOutputs._10a1_User_Data_128_bytes_1[82] := PlcOutputs._10a1_User_Data_128_bytes_1[82];
	HwOutputs._10a1_User_Data_128_bytes_1[83] := PlcOutputs._10a1_User_Data_128_bytes_1[83];
	HwOutputs._10a1_User_Data_128_bytes_1[84] := PlcOutputs._10a1_User_Data_128_bytes_1[84];
	HwOutputs._10a1_User_Data_128_bytes_1[85] := PlcOutputs._10a1_User_Data_128_bytes_1[85];
	HwOutputs._10a1_User_Data_128_bytes_1[86] := PlcOutputs._10a1_User_Data_128_bytes_1[86];
	HwOutputs._10a1_User_Data_128_bytes_1[87] := PlcOutputs._10a1_User_Data_128_bytes_1[87];
	HwOutputs._10a1_User_Data_128_bytes_1[88] := PlcOutputs._10a1_User_Data_128_bytes_1[88];
	HwOutputs._10a1_User_Data_128_bytes_1[89] := PlcOutputs._10a1_User_Data_128_bytes_1[89];
	HwOutputs._10a1_User_Data_128_bytes_1[90] := PlcOutputs._10a1_User_Data_128_bytes_1[90];
	HwOutputs._10a1_User_Data_128_bytes_1[91] := PlcOutputs._10a1_User_Data_128_bytes_1[91];
	HwOutputs._10a1_User_Data_128_bytes_1[92] := PlcOutputs._10a1_User_Data_128_bytes_1[92];
	HwOutputs._10a1_User_Data_128_bytes_1[93] := PlcOutputs._10a1_User_Data_128_bytes_1[93];
	HwOutputs._10a1_User_Data_128_bytes_1[94] := PlcOutputs._10a1_User_Data_128_bytes_1[94];
	HwOutputs._10a1_User_Data_128_bytes_1[95] := PlcOutputs._10a1_User_Data_128_bytes_1[95];
	HwOutputs._10a1_User_Data_128_bytes_1[96] := PlcOutputs._10a1_User_Data_128_bytes_1[96];
	HwOutputs._10a1_User_Data_128_bytes_1[97] := PlcOutputs._10a1_User_Data_128_bytes_1[97];
	HwOutputs._10a1_User_Data_128_bytes_1[98] := PlcOutputs._10a1_User_Data_128_bytes_1[98];
	HwOutputs._10a1_User_Data_128_bytes_1[99] := PlcOutputs._10a1_User_Data_128_bytes_1[99];
	HwOutputs._10a1_User_Data_128_bytes_1[100] := PlcOutputs._10a1_User_Data_128_bytes_1[100];
	HwOutputs._10a1_User_Data_128_bytes_1[101] := PlcOutputs._10a1_User_Data_128_bytes_1[101];
	HwOutputs._10a1_User_Data_128_bytes_1[102] := PlcOutputs._10a1_User_Data_128_bytes_1[102];
	HwOutputs._10a1_User_Data_128_bytes_1[103] := PlcOutputs._10a1_User_Data_128_bytes_1[103];
	HwOutputs._10a1_User_Data_128_bytes_1[104] := PlcOutputs._10a1_User_Data_128_bytes_1[104];
	HwOutputs._10a1_User_Data_128_bytes_1[105] := PlcOutputs._10a1_User_Data_128_bytes_1[105];
	HwOutputs._10a1_User_Data_128_bytes_1[106] := PlcOutputs._10a1_User_Data_128_bytes_1[106];
	HwOutputs._10a1_User_Data_128_bytes_1[107] := PlcOutputs._10a1_User_Data_128_bytes_1[107];
	HwOutputs._10a1_User_Data_128_bytes_1[108] := PlcOutputs._10a1_User_Data_128_bytes_1[108];
	HwOutputs._10a1_User_Data_128_bytes_1[109] := PlcOutputs._10a1_User_Data_128_bytes_1[109];
	HwOutputs._10a1_User_Data_128_bytes_1[110] := PlcOutputs._10a1_User_Data_128_bytes_1[110];
	HwOutputs._10a1_User_Data_128_bytes_1[111] := PlcOutputs._10a1_User_Data_128_bytes_1[111];
	HwOutputs._10a1_User_Data_128_bytes_1[112] := PlcOutputs._10a1_User_Data_128_bytes_1[112];
	HwOutputs._10a1_User_Data_128_bytes_1[113] := PlcOutputs._10a1_User_Data_128_bytes_1[113];
	HwOutputs._10a1_User_Data_128_bytes_1[114] := PlcOutputs._10a1_User_Data_128_bytes_1[114];
	HwOutputs._10a1_User_Data_128_bytes_1[115] := PlcOutputs._10a1_User_Data_128_bytes_1[115];
	HwOutputs._10a1_User_Data_128_bytes_1[116] := PlcOutputs._10a1_User_Data_128_bytes_1[116];
	HwOutputs._10a1_User_Data_128_bytes_1[117] := PlcOutputs._10a1_User_Data_128_bytes_1[117];
	HwOutputs._10a1_User_Data_128_bytes_1[118] := PlcOutputs._10a1_User_Data_128_bytes_1[118];
	HwOutputs._10a1_User_Data_128_bytes_1[119] := PlcOutputs._10a1_User_Data_128_bytes_1[119];
	HwOutputs._10a1_User_Data_128_bytes_1[120] := PlcOutputs._10a1_User_Data_128_bytes_1[120];
	HwOutputs._10a1_User_Data_128_bytes_1[121] := PlcOutputs._10a1_User_Data_128_bytes_1[121];
	HwOutputs._10a1_User_Data_128_bytes_1[122] := PlcOutputs._10a1_User_Data_128_bytes_1[122];
	HwOutputs._10a1_User_Data_128_bytes_1[123] := PlcOutputs._10a1_User_Data_128_bytes_1[123];
	HwOutputs._10a1_User_Data_128_bytes_1[124] := PlcOutputs._10a1_User_Data_128_bytes_1[124];
	HwOutputs._10a1_User_Data_128_bytes_1[125] := PlcOutputs._10a1_User_Data_128_bytes_1[125];
	HwOutputs._10a1_User_Data_128_bytes_1[126] := PlcOutputs._10a1_User_Data_128_bytes_1[126];
	HwOutputs._10a1_User_Data_128_bytes_1[127] := PlcOutputs._10a1_User_Data_128_bytes_1[127];
	HwOutputs._10a1_User_Data_128_bytes_1[128] := PlcOutputs._10a1_User_Data_128_bytes_1[128];
	HwOutputs._10a1_User_Data_128_bytes_1[129] := PlcOutputs._10a1_User_Data_128_bytes_1[129];
	HwOutputs._10a1_User_Data_128_bytes_1[130] := PlcOutputs._10a1_User_Data_128_bytes_1[130];
	HwOutputs._10a1_User_Data_128_bytes_1[131] := PlcOutputs._10a1_User_Data_128_bytes_1[131];
	HwOutputs.reader_st2_Acquisition_Control_1 := PlcOutputs.reader_st2_Acquisition_Control_1;
	HwOutputs.reader_st2_Results_Control_1 := PlcOutputs.reader_st2_Results_Control_1;
	HwOutputs.reader_st2_Soft_Event_Control_1 := PlcOutputs.reader_st2_Soft_Event_Control_1;
	HwOutputs.reader_st2_User_Data_64_bytes_1[0] := PlcOutputs.reader_st2_User_Data_64_bytes_1[0];
	HwOutputs.reader_st2_User_Data_64_bytes_1[1] := PlcOutputs.reader_st2_User_Data_64_bytes_1[1];
	HwOutputs.reader_st2_User_Data_64_bytes_1[2] := PlcOutputs.reader_st2_User_Data_64_bytes_1[2];
	HwOutputs.reader_st2_User_Data_64_bytes_1[3] := PlcOutputs.reader_st2_User_Data_64_bytes_1[3];
	HwOutputs.reader_st2_User_Data_64_bytes_1[4] := PlcOutputs.reader_st2_User_Data_64_bytes_1[4];
	HwOutputs.reader_st2_User_Data_64_bytes_1[5] := PlcOutputs.reader_st2_User_Data_64_bytes_1[5];
	HwOutputs.reader_st2_User_Data_64_bytes_1[6] := PlcOutputs.reader_st2_User_Data_64_bytes_1[6];
	HwOutputs.reader_st2_User_Data_64_bytes_1[7] := PlcOutputs.reader_st2_User_Data_64_bytes_1[7];
	HwOutputs.reader_st2_User_Data_64_bytes_1[8] := PlcOutputs.reader_st2_User_Data_64_bytes_1[8];
	HwOutputs.reader_st2_User_Data_64_bytes_1[9] := PlcOutputs.reader_st2_User_Data_64_bytes_1[9];
	HwOutputs.reader_st2_User_Data_64_bytes_1[10] := PlcOutputs.reader_st2_User_Data_64_bytes_1[10];
	HwOutputs.reader_st2_User_Data_64_bytes_1[11] := PlcOutputs.reader_st2_User_Data_64_bytes_1[11];
	HwOutputs.reader_st2_User_Data_64_bytes_1[12] := PlcOutputs.reader_st2_User_Data_64_bytes_1[12];
	HwOutputs.reader_st2_User_Data_64_bytes_1[13] := PlcOutputs.reader_st2_User_Data_64_bytes_1[13];
	HwOutputs.reader_st2_User_Data_64_bytes_1[14] := PlcOutputs.reader_st2_User_Data_64_bytes_1[14];
	HwOutputs.reader_st2_User_Data_64_bytes_1[15] := PlcOutputs.reader_st2_User_Data_64_bytes_1[15];
	HwOutputs.reader_st2_User_Data_64_bytes_1[16] := PlcOutputs.reader_st2_User_Data_64_bytes_1[16];
	HwOutputs.reader_st2_User_Data_64_bytes_1[17] := PlcOutputs.reader_st2_User_Data_64_bytes_1[17];
	HwOutputs.reader_st2_User_Data_64_bytes_1[18] := PlcOutputs.reader_st2_User_Data_64_bytes_1[18];
	HwOutputs.reader_st2_User_Data_64_bytes_1[19] := PlcOutputs.reader_st2_User_Data_64_bytes_1[19];
	HwOutputs.reader_st2_User_Data_64_bytes_1[20] := PlcOutputs.reader_st2_User_Data_64_bytes_1[20];
	HwOutputs.reader_st2_User_Data_64_bytes_1[21] := PlcOutputs.reader_st2_User_Data_64_bytes_1[21];
	HwOutputs.reader_st2_User_Data_64_bytes_1[22] := PlcOutputs.reader_st2_User_Data_64_bytes_1[22];
	HwOutputs.reader_st2_User_Data_64_bytes_1[23] := PlcOutputs.reader_st2_User_Data_64_bytes_1[23];
	HwOutputs.reader_st2_User_Data_64_bytes_1[24] := PlcOutputs.reader_st2_User_Data_64_bytes_1[24];
	HwOutputs.reader_st2_User_Data_64_bytes_1[25] := PlcOutputs.reader_st2_User_Data_64_bytes_1[25];
	HwOutputs.reader_st2_User_Data_64_bytes_1[26] := PlcOutputs.reader_st2_User_Data_64_bytes_1[26];
	HwOutputs.reader_st2_User_Data_64_bytes_1[27] := PlcOutputs.reader_st2_User_Data_64_bytes_1[27];
	HwOutputs.reader_st2_User_Data_64_bytes_1[28] := PlcOutputs.reader_st2_User_Data_64_bytes_1[28];
	HwOutputs.reader_st2_User_Data_64_bytes_1[29] := PlcOutputs.reader_st2_User_Data_64_bytes_1[29];
	HwOutputs.reader_st2_User_Data_64_bytes_1[30] := PlcOutputs.reader_st2_User_Data_64_bytes_1[30];
	HwOutputs.reader_st2_User_Data_64_bytes_1[31] := PlcOutputs.reader_st2_User_Data_64_bytes_1[31];
	HwOutputs.reader_st2_User_Data_64_bytes_1[32] := PlcOutputs.reader_st2_User_Data_64_bytes_1[32];
	HwOutputs.reader_st2_User_Data_64_bytes_1[33] := PlcOutputs.reader_st2_User_Data_64_bytes_1[33];
	HwOutputs.reader_st2_User_Data_64_bytes_1[34] := PlcOutputs.reader_st2_User_Data_64_bytes_1[34];
	HwOutputs.reader_st2_User_Data_64_bytes_1[35] := PlcOutputs.reader_st2_User_Data_64_bytes_1[35];
	HwOutputs.reader_st2_User_Data_64_bytes_1[36] := PlcOutputs.reader_st2_User_Data_64_bytes_1[36];
	HwOutputs.reader_st2_User_Data_64_bytes_1[37] := PlcOutputs.reader_st2_User_Data_64_bytes_1[37];
	HwOutputs.reader_st2_User_Data_64_bytes_1[38] := PlcOutputs.reader_st2_User_Data_64_bytes_1[38];
	HwOutputs.reader_st2_User_Data_64_bytes_1[39] := PlcOutputs.reader_st2_User_Data_64_bytes_1[39];
	HwOutputs.reader_st2_User_Data_64_bytes_1[40] := PlcOutputs.reader_st2_User_Data_64_bytes_1[40];
	HwOutputs.reader_st2_User_Data_64_bytes_1[41] := PlcOutputs.reader_st2_User_Data_64_bytes_1[41];
	HwOutputs.reader_st2_User_Data_64_bytes_1[42] := PlcOutputs.reader_st2_User_Data_64_bytes_1[42];
	HwOutputs.reader_st2_User_Data_64_bytes_1[43] := PlcOutputs.reader_st2_User_Data_64_bytes_1[43];
	HwOutputs.reader_st2_User_Data_64_bytes_1[44] := PlcOutputs.reader_st2_User_Data_64_bytes_1[44];
	HwOutputs.reader_st2_User_Data_64_bytes_1[45] := PlcOutputs.reader_st2_User_Data_64_bytes_1[45];
	HwOutputs.reader_st2_User_Data_64_bytes_1[46] := PlcOutputs.reader_st2_User_Data_64_bytes_1[46];
	HwOutputs.reader_st2_User_Data_64_bytes_1[47] := PlcOutputs.reader_st2_User_Data_64_bytes_1[47];
	HwOutputs.reader_st2_User_Data_64_bytes_1[48] := PlcOutputs.reader_st2_User_Data_64_bytes_1[48];
	HwOutputs.reader_st2_User_Data_64_bytes_1[49] := PlcOutputs.reader_st2_User_Data_64_bytes_1[49];
	HwOutputs.reader_st2_User_Data_64_bytes_1[50] := PlcOutputs.reader_st2_User_Data_64_bytes_1[50];
	HwOutputs.reader_st2_User_Data_64_bytes_1[51] := PlcOutputs.reader_st2_User_Data_64_bytes_1[51];
	HwOutputs.reader_st2_User_Data_64_bytes_1[52] := PlcOutputs.reader_st2_User_Data_64_bytes_1[52];
	HwOutputs.reader_st2_User_Data_64_bytes_1[53] := PlcOutputs.reader_st2_User_Data_64_bytes_1[53];
	HwOutputs.reader_st2_User_Data_64_bytes_1[54] := PlcOutputs.reader_st2_User_Data_64_bytes_1[54];
	HwOutputs.reader_st2_User_Data_64_bytes_1[55] := PlcOutputs.reader_st2_User_Data_64_bytes_1[55];
	HwOutputs.reader_st2_User_Data_64_bytes_1[56] := PlcOutputs.reader_st2_User_Data_64_bytes_1[56];
	HwOutputs.reader_st2_User_Data_64_bytes_1[57] := PlcOutputs.reader_st2_User_Data_64_bytes_1[57];
	HwOutputs.reader_st2_User_Data_64_bytes_1[58] := PlcOutputs.reader_st2_User_Data_64_bytes_1[58];
	HwOutputs.reader_st2_User_Data_64_bytes_1[59] := PlcOutputs.reader_st2_User_Data_64_bytes_1[59];
	HwOutputs.reader_st2_User_Data_64_bytes_1[60] := PlcOutputs.reader_st2_User_Data_64_bytes_1[60];
	HwOutputs.reader_st2_User_Data_64_bytes_1[61] := PlcOutputs.reader_st2_User_Data_64_bytes_1[61];
	HwOutputs.reader_st2_User_Data_64_bytes_1[62] := PlcOutputs.reader_st2_User_Data_64_bytes_1[62];
	HwOutputs.reader_st2_User_Data_64_bytes_1[63] := PlcOutputs.reader_st2_User_Data_64_bytes_1[63];
	HwOutputs.reader_st2_User_Data_64_bytes_1[64] := PlcOutputs.reader_st2_User_Data_64_bytes_1[64];
	HwOutputs.reader_st2_User_Data_64_bytes_1[65] := PlcOutputs.reader_st2_User_Data_64_bytes_1[65];
	HwOutputs.reader_st2_User_Data_64_bytes_1[66] := PlcOutputs.reader_st2_User_Data_64_bytes_1[66];
	HwOutputs.reader_st2_User_Data_64_bytes_1[67] := PlcOutputs.reader_st2_User_Data_64_bytes_1[67];
	// HwOutputs._7600_Acquisition_Control_1 := PlcOutputs._7600_Acquisition_Control_1;
	// HwOutputs._7600_Inspection_Control_1 := PlcOutputs._7600_Inspection_Control_1;
	// HwOutputs._7600_Command_Control_1 := PlcOutputs._7600_Command_Control_1;
	// HwOutputs._7600_SoftEvent_Control_1 := PlcOutputs._7600_SoftEvent_Control_1;
	// HwOutputs._7600_User_Data_64_bytes_1[0] := PlcOutputs._7600_User_Data_64_bytes_1[0];
	// HwOutputs._7600_User_Data_64_bytes_1[1] := PlcOutputs._7600_User_Data_64_bytes_1[1];
	// HwOutputs._7600_User_Data_64_bytes_1[2] := PlcOutputs._7600_User_Data_64_bytes_1[2];
	// HwOutputs._7600_User_Data_64_bytes_1[3] := PlcOutputs._7600_User_Data_64_bytes_1[3];
	// HwOutputs._7600_User_Data_64_bytes_1[4] := PlcOutputs._7600_User_Data_64_bytes_1[4];
	// HwOutputs._7600_User_Data_64_bytes_1[5] := PlcOutputs._7600_User_Data_64_bytes_1[5];
	// HwOutputs._7600_User_Data_64_bytes_1[6] := PlcOutputs._7600_User_Data_64_bytes_1[6];
	// HwOutputs._7600_User_Data_64_bytes_1[7] := PlcOutputs._7600_User_Data_64_bytes_1[7];
	// HwOutputs._7600_User_Data_64_bytes_1[8] := PlcOutputs._7600_User_Data_64_bytes_1[8];
	// HwOutputs._7600_User_Data_64_bytes_1[9] := PlcOutputs._7600_User_Data_64_bytes_1[9];
	// HwOutputs._7600_User_Data_64_bytes_1[10] := PlcOutputs._7600_User_Data_64_bytes_1[10];
	// HwOutputs._7600_User_Data_64_bytes_1[11] := PlcOutputs._7600_User_Data_64_bytes_1[11];
	// HwOutputs._7600_User_Data_64_bytes_1[12] := PlcOutputs._7600_User_Data_64_bytes_1[12];
	// HwOutputs._7600_User_Data_64_bytes_1[13] := PlcOutputs._7600_User_Data_64_bytes_1[13];
	// HwOutputs._7600_User_Data_64_bytes_1[14] := PlcOutputs._7600_User_Data_64_bytes_1[14];
	// HwOutputs._7600_User_Data_64_bytes_1[15] := PlcOutputs._7600_User_Data_64_bytes_1[15];
	// HwOutputs._7600_User_Data_64_bytes_1[16] := PlcOutputs._7600_User_Data_64_bytes_1[16];
	// HwOutputs._7600_User_Data_64_bytes_1[17] := PlcOutputs._7600_User_Data_64_bytes_1[17];
	// HwOutputs._7600_User_Data_64_bytes_1[18] := PlcOutputs._7600_User_Data_64_bytes_1[18];
	// HwOutputs._7600_User_Data_64_bytes_1[19] := PlcOutputs._7600_User_Data_64_bytes_1[19];
	// HwOutputs._7600_User_Data_64_bytes_1[20] := PlcOutputs._7600_User_Data_64_bytes_1[20];
	// HwOutputs._7600_User_Data_64_bytes_1[21] := PlcOutputs._7600_User_Data_64_bytes_1[21];
	// HwOutputs._7600_User_Data_64_bytes_1[22] := PlcOutputs._7600_User_Data_64_bytes_1[22];
	// HwOutputs._7600_User_Data_64_bytes_1[23] := PlcOutputs._7600_User_Data_64_bytes_1[23];
	// HwOutputs._7600_User_Data_64_bytes_1[24] := PlcOutputs._7600_User_Data_64_bytes_1[24];
	// HwOutputs._7600_User_Data_64_bytes_1[25] := PlcOutputs._7600_User_Data_64_bytes_1[25];
	// HwOutputs._7600_User_Data_64_bytes_1[26] := PlcOutputs._7600_User_Data_64_bytes_1[26];
	// HwOutputs._7600_User_Data_64_bytes_1[27] := PlcOutputs._7600_User_Data_64_bytes_1[27];
	// HwOutputs._7600_User_Data_64_bytes_1[28] := PlcOutputs._7600_User_Data_64_bytes_1[28];
	// HwOutputs._7600_User_Data_64_bytes_1[29] := PlcOutputs._7600_User_Data_64_bytes_1[29];
	// HwOutputs._7600_User_Data_64_bytes_1[30] := PlcOutputs._7600_User_Data_64_bytes_1[30];
	// HwOutputs._7600_User_Data_64_bytes_1[31] := PlcOutputs._7600_User_Data_64_bytes_1[31];
	// HwOutputs._7600_User_Data_64_bytes_1[32] := PlcOutputs._7600_User_Data_64_bytes_1[32];
	// HwOutputs._7600_User_Data_64_bytes_1[33] := PlcOutputs._7600_User_Data_64_bytes_1[33];
	// HwOutputs._7600_User_Data_64_bytes_1[34] := PlcOutputs._7600_User_Data_64_bytes_1[34];
	// HwOutputs._7600_User_Data_64_bytes_1[35] := PlcOutputs._7600_User_Data_64_bytes_1[35];
	// HwOutputs._7600_User_Data_64_bytes_1[36] := PlcOutputs._7600_User_Data_64_bytes_1[36];
	// HwOutputs._7600_User_Data_64_bytes_1[37] := PlcOutputs._7600_User_Data_64_bytes_1[37];
	// HwOutputs._7600_User_Data_64_bytes_1[38] := PlcOutputs._7600_User_Data_64_bytes_1[38];
	// HwOutputs._7600_User_Data_64_bytes_1[39] := PlcOutputs._7600_User_Data_64_bytes_1[39];
	// HwOutputs._7600_User_Data_64_bytes_1[40] := PlcOutputs._7600_User_Data_64_bytes_1[40];
	// HwOutputs._7600_User_Data_64_bytes_1[41] := PlcOutputs._7600_User_Data_64_bytes_1[41];
	// HwOutputs._7600_User_Data_64_bytes_1[42] := PlcOutputs._7600_User_Data_64_bytes_1[42];
	// HwOutputs._7600_User_Data_64_bytes_1[43] := PlcOutputs._7600_User_Data_64_bytes_1[43];
	// HwOutputs._7600_User_Data_64_bytes_1[44] := PlcOutputs._7600_User_Data_64_bytes_1[44];
	// HwOutputs._7600_User_Data_64_bytes_1[45] := PlcOutputs._7600_User_Data_64_bytes_1[45];
	// HwOutputs._7600_User_Data_64_bytes_1[46] := PlcOutputs._7600_User_Data_64_bytes_1[46];
	// HwOutputs._7600_User_Data_64_bytes_1[47] := PlcOutputs._7600_User_Data_64_bytes_1[47];
	// HwOutputs._7600_User_Data_64_bytes_1[48] := PlcOutputs._7600_User_Data_64_bytes_1[48];
	// HwOutputs._7600_User_Data_64_bytes_1[49] := PlcOutputs._7600_User_Data_64_bytes_1[49];
	// HwOutputs._7600_User_Data_64_bytes_1[50] := PlcOutputs._7600_User_Data_64_bytes_1[50];
	// HwOutputs._7600_User_Data_64_bytes_1[51] := PlcOutputs._7600_User_Data_64_bytes_1[51];
	// HwOutputs._7600_User_Data_64_bytes_1[52] := PlcOutputs._7600_User_Data_64_bytes_1[52];
	// HwOutputs._7600_User_Data_64_bytes_1[53] := PlcOutputs._7600_User_Data_64_bytes_1[53];
	// HwOutputs._7600_User_Data_64_bytes_1[54] := PlcOutputs._7600_User_Data_64_bytes_1[54];
	// HwOutputs._7600_User_Data_64_bytes_1[55] := PlcOutputs._7600_User_Data_64_bytes_1[55];
	// HwOutputs._7600_User_Data_64_bytes_1[56] := PlcOutputs._7600_User_Data_64_bytes_1[56];
	// HwOutputs._7600_User_Data_64_bytes_1[57] := PlcOutputs._7600_User_Data_64_bytes_1[57];
	// HwOutputs._7600_User_Data_64_bytes_1[58] := PlcOutputs._7600_User_Data_64_bytes_1[58];
	// HwOutputs._7600_User_Data_64_bytes_1[59] := PlcOutputs._7600_User_Data_64_bytes_1[59];
	// HwOutputs._7600_User_Data_64_bytes_1[60] := PlcOutputs._7600_User_Data_64_bytes_1[60];
	// HwOutputs._7600_User_Data_64_bytes_1[61] := PlcOutputs._7600_User_Data_64_bytes_1[61];
	// HwOutputs._7600_User_Data_64_bytes_1[62] := PlcOutputs._7600_User_Data_64_bytes_1[62];
	// HwOutputs._7600_User_Data_64_bytes_1[63] := PlcOutputs._7600_User_Data_64_bytes_1[63];
END_FUNCTION
